(* IEC 61131-3 sources: programs/VI-54/VI-54_20171205/VI-54_20171205/Stations/PLC_VI54/VI-54_171014/Class/TestTrigger, 1 file *)

(* ---- TestTrigger.st ---- *)
(*!
<Class
	Name               = "TestTrigger"
	Revision           = "1.1"
	RealtimeTask       = "false"
	CyclicTask         = "false"
	BackgroundTask     = "false"
	Sigmatek           = "false"
	OSInterface        = "false"
	HighPriority       = "false"
	Automatic          = "false"
	UpdateMode         = "Prescan"
	SharedCommandTable = "true"
	Objectsize         = "(510,240)">
	<Channels>
		<Server Name="ProdsPerMin" Visualized="true" Initialize="false" WriteProtected="false" Retentive="File"/>
		<Server Name="TestTriggerOn" Visualized="true" Initialize="false" WriteProtected="false" Retentive="false"/>
		<Server Name="Trigger" Visualized="true" Initialize="false" WriteProtected="true" Retentive="false"/>
		<Client Name="iExtTrigger" Required="false" Internal="false"/>
		<Client Name="iFcTrigger" Required="true" Internal="false"/>
		<Client Name="LMC_Axle" Required="false" Internal="false"/>
		<Client Name="STD" Required="true" Internal="true"/>
	</Channels>
	<Network Name="TestTrigger">
		<!-- List of Components in this network -->
		<Components>
			<Object
				Name           = "STD"
				Class          = "Standard"
				Position       = "(210,360)"
				Visualized     = "false"
				BackgroundTime = "1000 ms">
				<Channels>
					<Server Name="ClassSvr"/>
				</Channels>
			</Object>
		</Components>
		<Comments>
		</Comments>
		<!-- List of Connections in this network -->
		<Connections>
			<Connection Source="this.STD" Destination="STD.ClassSvr"/>
		</Connections>
		<!-- Headerfiles -->
		<Options>
		</Options>
	</Network>
</Class>
*)
TestTrigger : CLASS
  //Servers:
	Trigger 	: SvrChCmd_DINT;
	TestTriggerOn 	: SvrCh_DINT;
	ProdsPerMin 	: SvrCh_DINT;
  //Clients:
	iFcTrigger 	: CltCh_DINT;
	iExtTrigger 	: CltCh_DINT;
	LMC_Axle 	: CltChCmd__LMCAxis;
	STD 	: CltChCmd_Standard;
  //Variables:
		Time_ms 	: UDINT;
		TmrMaintrigger 	: UDINT;
		TriggerBits : BDINT
		[
		  1 Active,
		];

  //Functions:

	FUNCTION VIRTUAL GLOBAL Trigger::Read
		VAR_OUTPUT
			output (EAX) 	: DINT;
		END_VAR;
  //Tables:
	FUNCTION @STD
		VAR_OUTPUT
			ret_code	: CONFSTATES;
		END_VAR;
	FUNCTION GLOBAL TAB @CT_;
END_CLASS;

#pragma using Standard
#pragma usingLtd _LMCAxis

FUNCTION VIRTUAL GLOBAL TestTrigger::Trigger::Read
	VAR_OUTPUT
		output (EAX) 	: DINT;
	END_VAR

  // Read external input
  if IsClientConnected(#iExtTrigger) then
    iExtTrigger := iExtTrigger.Read();
  end_if;
  iFcTrigger := iFcTrigger.Read();

  // Check of LMC is moving
  if LMC_Axle.ActVelocity > 0 then
    TriggerBits.Active := True;
  else
    TriggerBits.Active := False;
  end_if;

  // Calculate time interface
  if ProdsPerMin > 0 then
    Time_ms := 60000 / (to_udint ProdsPerMin);  // omzetten naar ms
  else
    Time_ms := 60000;
  end_if;

  if TriggerBits.Active = 1 then
    if TestTriggerOn = 1 then
      if ops.tAbsolute - TmrMaintrigger >= Time_ms then
        Trigger := 1;
        TmrMaintrigger := ops.tAbsolute;
      end_if;
      if STD.TON(IN:= Trigger, PT:= 20) then
        Trigger := 0;
      end_if;
    else
      Trigger := (iFcTrigger = 1 | iExtTrigger = 1);
    end_if;
  else
    Trigger := 0;
  end_if;

	output := Trigger;

END_FUNCTION
